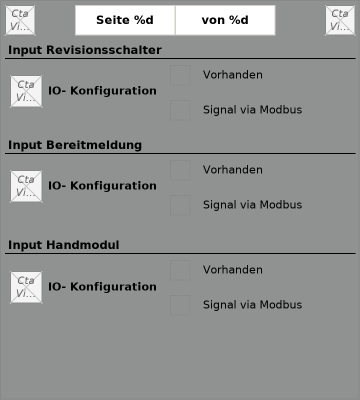
VISUALIZATION StellAntrieb_ParameterIO  // 360x400
VAR_INPUT
    ITF_STELLANTRIEBIN : ITF_STELLANTRIEB;
END_VAR
VAR
    uiPage  :   UINT;
    uiMin   :   UINT    := 0;
    uiMax   :   UINT    := 4;
END_VAR
    Frame (0,40 360x360), frame switch variable: uiPage
        shows StellAntrieb_ParameterIO0(ITF_STELLANTRIEBIN := ITF_STELLANTRIEBIN, ITF_RevSwitch_IN := ITF_STELLANTRIEBIN.proRevisionSwitch_ITF, ITF_Ready_IN := ITF_STELLANTRIEBIN.proActuatorReady_ITF, ITF_HandModul_IN := ITF_STELLANTRIEBIN.proHandModul_ITF)
        shows StellAntrieb_ParameterIO1(ITF_STELLANTRIEBIN := ITF_STELLANTRIEBIN, ITF_RückClosed_IN := ITF_STELLANTRIEBIN.proIsClosed_ITF)
        shows StellAntrieb_ParameterIO2(ITF_STELLANTRIEBIN := ITF_STELLANTRIEBIN, ITF_RückOffen_IN := ITF_STELLANTRIEBIN.proIsOpen_ITF)
        shows StellAntrieb_ParameterIO3(ITF_STELLANTRIEBIN := ITF_STELLANTRIEBIN, ITF_ActualPos_IN := ITF_STELLANTRIEBIN.proActualPosition_ITF)
        shows StellAntrieb_ParameterIO4(ITF_STELLANTRIEBIN := ITF_STELLANTRIEBIN, ITF_xOnAuf_IN := ITF_STELLANTRIEBIN.proOnOpen_ITF, ITF_xOnZu_IN := ITF_STELLANTRIEBIN.proOnClose_ITF, ITF_rOnY_IN := ITF_STELLANTRIEBIN.proOnY_ITF)
    Image (325,5 30x30), invisible if: uiPage = uiMax, image: CtaVisSymbols.ImagePool.arrow-right_square
        OnMouseClick: execute {
            uiPage := uiPage + 1;
            IF uiPage >= uiMax THEN
                uiPage := uiMax;
            END_IF;
        }
    Image (5,5 30x30), invisible if: uiPage = uiMin, image: CtaVisSymbols.ImagePool.arrow-left_square
        OnMouseClick: execute {
            uiPage := uiPage - 1;
            IF uiPage <= uiMin THEN
                uiPage := uiMin;
            END_IF;
        }
    Textfield (175,5 100x30), "von %d", text variable: uiMax
    Textfield (75,5 100x30), "Seite %d", text variable: uiPage
END_VISUALIZATION

// 40 Visualizations/POPUP/PARAMETER/StellAntrieb_IO/StellAntrieb_ParameterIO2
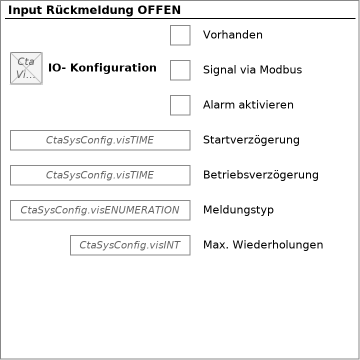
VISUALIZATION StellAntrieb_ParameterIO2  // 360x360
VAR_INPUT
    ITF_STELLANTRIEBIN 	:	ITF_STELLANTRIEB;
	ITF_RückOffen_IN	:	CtaSysIO.ITF_IO;
END_VAR
    Label (5,0 350x20), "Input Rückmeldung OFFEN"
    Frame (170,25 20x20)
        shows CtaSysConfig.visBOOL(visfbBOOLIn := ITF_STELLANTRIEBIN.p_scInStellAtRükOpen_fbxEnable)
    Label (200,25 150x20), "Vorhanden"
    Frame (170,60 20x20)
        shows CtaSysConfig.visBOOL(visfbBOOLIn := ITF_STELLANTRIEBIN.p_scInStellAtRükOpen_fbxInputMb)
    Label (200,60 150x20), "Signal via Modbus"
    Frame (170,95 20x20)
        shows CtaSysConfig.visBOOL(visfbBOOLIn := ITF_STELLANTRIEBIN.p_scInStellAtRükOpen_fbxDoesAlarm)
    Label (200,95 150x20), "Alarm aktivieren"
    Frame (10,130 180x20)
        shows CtaSysConfig.visTIME(visfbTIMEIn := ITF_STELLANTRIEBIN.p_scInStellAtRükOpen_fbtDelayStart)
    Label (200,130 150x20), "Startverzögerung"
    Label (200,165 150x20), "Betriebsverzögerung"
    Frame (10,165 180x20)
        shows CtaSysConfig.visTIME(visfbTIMEIn := ITF_STELLANTRIEBIN.p_scInStellAtRükOpen_fbtDelayRun)
    Label (200,200 150x20), "Meldungstyp"
    Label (200,235 150x20), "Max. Wiederholungen"
    Line (5,18) (355,18)
    Frame (10,200 180x20), text list: 'CtaAppReport.txtLibAp99_2enTypeOfAck', text index: CtaSysConfig.fcGetEnumerationId(ITF_STELLANTRIEBIN.p_scInStellAtRükOpen_fbiTypeOfAck)
        shows CtaSysConfig.visENUMERATION(visfbENUIn := ITF_STELLANTRIEBIN.p_scInStellAtRükOpen_fbiTypeOfAck)
    Frame (70,235 120x20)
        shows CtaSysConfig.visINT(visfbINTIn := ITF_STELLANTRIEBIN.p_scInStellAtRükOpen_fbiMaxErrorRetryAllowed)
    Image (10,52 32x32), invisible if: ITF_RückOffen_IN = 0, image: CtaVisSymbols.ImagePool.build
        OnMouseDown:  Dialog=StellAntrieb_POPUP_IO_ITF, Parameters={ITF_IO_IN: ITF_RückOffen_IN}, OpenModal=True, OpenCentered=True
    Label (45,58 120x20), "IO- Konfiguration", invisible if: ITF_RückOffen_IN = 0
END_VISUALIZATION

// 40 Visualizations/POPUP/PARAMETER/StellAntrieb_IO/StellAntrieb_ParameterIO3
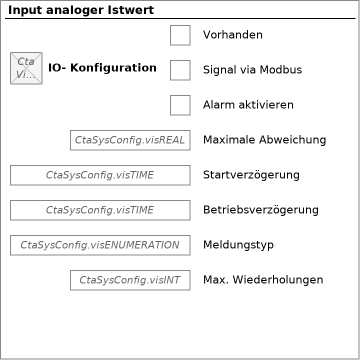
VISUALIZATION StellAntrieb_ParameterIO3  // 360x360
VAR_INPUT
    ITF_STELLANTRIEBIN 	:	ITF_STELLANTRIEB;
	ITF_ActualPos_IN	:	CtaSysIO.ITF_IO;
END_VAR
    Label (5,0 350x20), "Input analoger Istwert"
    Frame (170,25 20x20)
        shows CtaSysConfig.visBOOL(visfbBOOLIn := ITF_STELLANTRIEBIN.p_scInStellAtActualPosition_fbxEnable)
    Label (200,25 150x20), "Vorhanden"
    Frame (170,60 20x20)
        shows CtaSysConfig.visBOOL(visfbBOOLIn := ITF_STELLANTRIEBIN.p_scInStellAtActualPosition_fbxInputMb)
    Label (200,60 150x20), "Signal via Modbus"
    Frame (170,95 20x20)
        shows CtaSysConfig.visBOOL(visfbBOOLIn := ITF_STELLANTRIEBIN.p_scInStellAtActualPosition_fbxDoesAlarm)
    Label (200,95 150x20), "Alarm aktivieren"
    Frame (10,165 180x20)
        shows CtaSysConfig.visTIME(visfbTIMEIn := ITF_STELLANTRIEBIN.p_scInStellAtActualPosition_fbtDelayStart)
    Label (200,165 150x20), "Startverzögerung"
    Label (200,200 150x20), "Betriebsverzögerung"
    Frame (10,200 180x20)
        shows CtaSysConfig.visTIME(visfbTIMEIn := ITF_STELLANTRIEBIN.p_scInStellAtActualPosition_fbtDelayRun)
    Frame (70,130 120x20)
        shows CtaSysConfig.visREAL(visfbREALIn := ITF_STELLANTRIEBIN.p_scInStellAtActualPosition_fbrMaxDiff, stPhysikalischeEinheit := '%')
    Label (200,130 150x20), "Maximale Abweichung"
    Label (200,235 150x20), "Meldungstyp"
    Label (200,270 150x20), "Max. Wiederholungen"
    Line (5,18) (355,18)
    Frame (10,235 180x20), text list: 'CtaAppReport.txtLibAp99_2enTypeOfAck', text index: CtaSysConfig.fcGetEnumerationId(ITF_STELLANTRIEBIN.p_scInStellAtActualPosition_fbiTypeOfAck)
        shows CtaSysConfig.visENUMERATION(visfbENUIn := ITF_STELLANTRIEBIN.p_scInStellAtActualPosition_fbiTypeOfAck)
    Frame (70,270 120x20)
        shows CtaSysConfig.visINT(visfbINTIn := ITF_STELLANTRIEBIN.p_scInStellAtActualPosition_fbiMaxErrorRetryAllowed)
    Label (45,58 120x20), "IO- Konfiguration", invisible if: ITF_ActualPos_IN = 0
    Image (10,52 32x32), invisible if: ITF_ActualPos_IN = 0, image: CtaVisSymbols.ImagePool.build
        OnMouseDown:  Dialog=StellAntrieb_POPUP_IO_ITF, Parameters={ITF_IO_IN: ITF_ActualPos_IN}, OpenModal=True, OpenCentered=True
END_VISUALIZATION

// 40 Visualizations/POPUP/PARAMETER/StellAntrieb_InfluxDb/StellAntrieb_ParameterInfluxDb
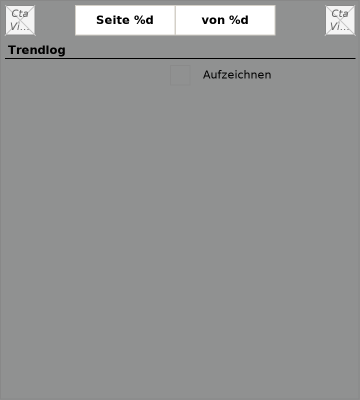
VISUALIZATION StellAntrieb_ParameterInfluxDb  // 360x400
VAR_INPUT
    ITF_STELLANTRIEBIN : ITF_STELLANTRIEB;
END_VAR
VAR
    uiPage  :   UINT;
    uiMin   :   UINT    := 0;
    uiMax   :   UINT    := 0;
END_VAR
    Image (5,5 30x30), invisible if: uiPage = uiMin, image: CtaVisSymbols.ImagePool.arrow-left_square
        OnMouseClick: execute {
            uiPage := uiPage - 1;
            IF uiPage <= uiMin THEN
                uiPage := uiMin;
            END_IF;
        }
    Image (325,5 30x30), invisible if: uiPage = uiMax, image: CtaVisSymbols.ImagePool.arrow-right_square
        OnMouseClick: execute {
            uiPage := uiPage + 1;
            IF uiPage >= uiMax THEN
                uiPage := uiMax;
            END_IF;
        }
    Frame (0,40 360x360), frame switch variable: uiPage
        shows StellAntrieb_ParameterInfluxDb0(ITF_STELLANTRIEBIN := ITF_STELLANTRIEBIN)
        shows AT_ParameterIO1(ITF_Parameter := ITF_Parameter)
        pReferences[0]: ITF_Parameter=ITF_Parameter
    Textfield (75,5 100x30), "Seite %d", text variable: uiPage
    Textfield (175,5 100x30), "von %d", text variable: uiMax
END_VISUALIZATION

// 40 Visualizations/POPUP/PARAMETER/StellAntrieb_InfluxDb/StellAntrieb_ParameterInfluxDb0
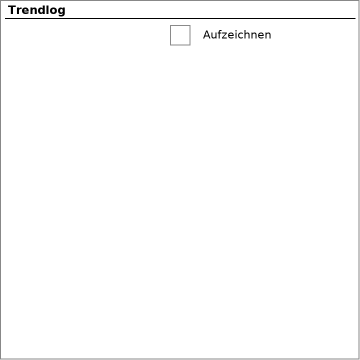
VISUALIZATION StellAntrieb_ParameterInfluxDb0  // 360x360
VAR_INPUT
    ITF_STELLANTRIEBIN : ITF_STELLANTRIEB;
END_VAR
    Frame (170,25 20x20)
        shows CtaSysConfig.visBOOL(visfbBOOLIn := ITF_STELLANTRIEBIN.p_scInfluxDb_fbxEnable)
    Label (200,25 150x20), "Aufzeichnen"
    Label (5,0 350x20), "Trendlog"
    Line (5,18) (355,18)
END_VISUALIZATION

// 40 Visualizations/POPUP/IO/StellAntrieb_IO0
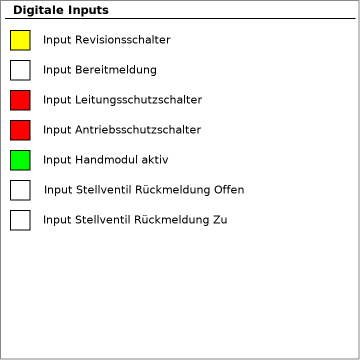
VISUALIZATION StellAntrieb_IO0  // 360x360
VAR_INPUT
    ITF_STELLANTRIEBIN    :   ITF_STELLANTRIEB;	
END_VAR
    Label (40,30 320x20), "Input Revisionsschalter", invisible if: ITF_STELLANTRIEBIN.proNotShowDI_RevisionSwitchOk
    Label (40,60 320x20), "Input Bereitmeldung", invisible if: ITF_STELLANTRIEBIN.proNotShowDI_Ready
    Rectangle (10,30 20x20), colour toggle: ITF_STELLANTRIEBIN.proGetDI_RevisionSwitchOK, invisible if: ITF_STELLANTRIEBIN.proNotShowDI_RevisionSwitchOk
    Rectangle (10,60 20x20), colour toggle: ITF_STELLANTRIEBIN.proGetDI_IsReady, invisible if: ITF_STELLANTRIEBIN.proNotShowDI_Ready
    Rectangle (10,90 20x20), colour toggle: ITF_STELLANTRIEBIN.proGetDI_FuseOK, invisible if: ITF_STELLANTRIEBIN.proNotShowDI_FuseOk
    Label (40,90 320x20), "Input Leitungsschutzschalter", invisible if: ITF_STELLANTRIEBIN.proNotShowDI_FuseOk
    Label (40,120 320x20), "Input Antriebsschutzschalter", invisible if: ITF_STELLANTRIEBIN.proNotShowDI_ActuatorFuseOk
    Rectangle (10,120 20x20), colour toggle: ITF_STELLANTRIEBIN.proGetDI_ActuatorFuseOk, invisible if: ITF_STELLANTRIEBIN.proNotShowDI_ActuatorFuseOk
    Label (40,150 320x20), "Input Handmodul aktiv", invisible if: ITF_STELLANTRIEBIN.proNotShowDI_ActuatorHand
    Rectangle (10,150 20x20), colour toggle: ITF_STELLANTRIEBIN.proGetDI_ActuatorHand, invisible if: ITF_STELLANTRIEBIN.proNotShowDI_ActuatorHand
    Label (10,0 350x20), "Digitale Inputs"
    Rectangle (10,210 20x20), colour toggle: ITF_STELLANTRIEBIN.proGetDI_RükIsClosed, invisible if: ITF_STELLANTRIEBIN.proNotShowDI_RükIsOpen
    Label (40,210 320x20), "Input Stellventil Rückmeldung Zu", invisible if: ITF_STELLANTRIEBIN.proNotShowDI_RükIsOpen
    Rectangle (10,180 20x20), colour toggle: ITF_STELLANTRIEBIN.proGetDI_RükIsOpen, invisible if: ITF_STELLANTRIEBIN.proNotShowDI_RükIsOpen
    Label (41,180 320x20), "Input Stellventil Rückmeldung Offen", invisible if: ITF_STELLANTRIEBIN.proNotShowDI_RükIsOpen
    Line (5,18) (355,18)
END_VISUALIZATION

// 40 Visualizations/POPUP/IO/StellAntrieb_IO
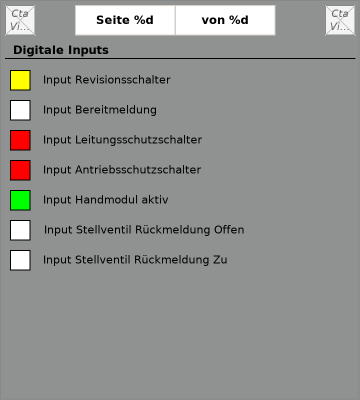
VISUALIZATION StellAntrieb_IO  // 360x400
VAR_INPUT
    ITF_STELLANTRIEBIN    :   ITF_STELLANTRIEB;	
END_VAR
VAR
    uiPage  :   UINT;
    uiMin   :   UINT    := 0;
    uiMax   :   UINT    := 1;
END_VAR
    Frame (0,40 360x360), frame switch variable: uiPage
        shows StellAntrieb_IO0(ITF_STELLANTRIEBIN := ITF_STELLANTRIEBIN)
        shows StellAntrieb_IO1(ITF_STELLANTRIEBIN := ITF_STELLANTRIEBIN)
        shows AT_ParameterIO2(ITF_Parameter := ITF_Parameter)
        shows AT_ParameterIO3(ITF_Parameter := ITF_Parameter)
    Image (325,5 30x30), invisible if: uiPage = uiMax, image: CtaVisSymbols.ImagePool.arrow-right_square
        OnMouseClick: execute {
            uiPage := uiPage + 1;
            IF uiPage >= uiMax THEN
                uiPage := uiMax;
            END_IF;
        }
    Image (5,5 30x30), invisible if: uiPage = uiMin, image: CtaVisSymbols.ImagePool.arrow-left_square
        OnMouseClick: execute {
            uiPage := uiPage - 1;
            IF uiPage <= uiMin THEN
                uiPage := uiMin;
            END_IF;
        }
    Textfield (175,5 100x30), "von %d", text variable: uiMax
    Textfield (75,5 100x30), "Seite %d", text variable: uiPage
END_VISUALIZATION

// 40 Visualizations/POPUP/IO/StellAntrieb_IO1
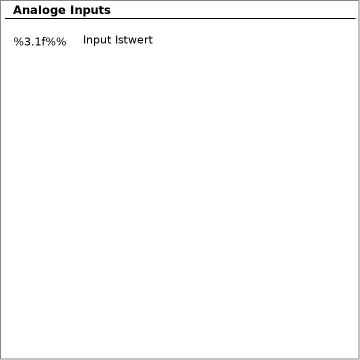
VISUALIZATION StellAntrieb_IO1  // 360x360
VAR_INPUT
    ITF_STELLANTRIEBIN    :   ITF_STELLANTRIEB;	
END_VAR
    Label (80,30 280x20), "Input Istwert", invisible if: ITF_STELLANTRIEBIN.proNotShowAI_ActualPosition
    Label (10,0 350x20), "Analoge Inputs"
    Textfield (10,32 60x20), "%3.1f%%", text variable: ITF_STELLANTRIEBIN.proGetAI_ActualPosition, invisible if: ITF_STELLANTRIEBIN.proNotShowAI_ActualPosition
    Line (5,18) (355,18)
END_VISUALIZATION

// 40 Visualizations/ICON/StellAntrieb_BASE/Ventile/DurchflussVentil/Motor_Left/ML_Durchgang
VISUALIZATION ML_Durchgang  // 15x30
VAR_INPUT
	rProzent	:	REAL;
END_VAR
    Line (0,15) (8,15)
    Polygon (8,15) (15,0) (0,0)
    Polygon (8,15) (15,30) (0,30)
    Polygon (8,15) (15,0) (0,0)
        p1097714728: fcValveAnimation(rProzent,TRUE)
END_VISUALIZATION

// 40 Visualizations/ICON/StellAntrieb_BASE/Icons/Motor_Left/Icon_ML_AB_Down
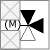
VISUALIZATION Icon_ML_AB_Down  // 50x50
VAR_INPUT
    ITF_STELLANTRIEB_IN   :   ITF_STELLANTRIEB;	
END_VAR
    Frame (5,17 15x15)
        shows Motor(ITF_STELLANTRIEB_IN := ITF_STELLANTRIEB_IN)
    Frame (20,10 22x30)
        shows ML_Ventil_AB_Down(rProzent := ITF_STELLANTRIEB_IN.proOnY)
    Image (0,0 20x20), invisible if: NOT ITF_STELLANTRIEB_IN.proIsWarning, image: CtaVisSymbols.ImagePool.CtaWarning
    Image (0,30 20x20), invisible if: NOT ITF_STELLANTRIEB_IN.proIsHandOnOrOff, image: CtaVisSymbols.ImagePool.front_hand_Yellow
    Image (0,30 20x20), invisible if: NOT ITF_STELLANTRIEB_IN.proHandOff, image: CtaVisSymbols.ImagePool.front_hand_Yellow_Off
END_VISUALIZATION

// 40 Visualizations/ICON/StellAntrieb_BASE/Ventile/DreiWegVentil/Motor_Above/MA_Ventil_AB_L
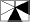
VISUALIZATION MA_Ventil_AB_L  // 30x22
VAR_INPUT
	rProzent	:	REAL;
END_VAR
    Polygon (0,0) (15,7) (0,15)
    Polygon (15,7) (22,22) (7,22)
    Polygon (15,7) (30,0) (30,15)
    Line (15,7) (15,0)
    Polygon (15,7) (30,0) (30,15)
        p1097714728: fcValveAnimation(rProzent,TRUE)
    Polygon (15,7) (22,22) (7,22)
        p1097714728: fcValveAnimation(rProzent,FALSE)
END_VISUALIZATION

// 40 Visualizations/ICON/StellAntrieb_BASE/Ventile/DreiWegVentil/Motor_Above/MA_Ventil_Verteiler
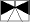
VISUALIZATION MA_Ventil_Verteiler  // 30x22
VAR_INPUT
	rProzent	:	REAL;
END_VAR
    Polygon (0,0) (15,7) (0,15)
    Polygon (15,7) (22,22) (7,22)
    Polygon (15,7) (30,0) (30,15)
    Line (15,7) (15,0)
    Polygon (15,7) (30,0) (30,15)
        p1097714728: fcValveAnimation(rProzent,FALSE)
    Polygon (0,0) (15,7) (0,15)
        p1097714728: fcValveAnimation(rProzent,TRUE)
END_VISUALIZATION

// 40 Visualizations/ICON/StellAntrieb_BASE/Ventile/DreiWegVentil/Motor_Above/MA_Ventil_AB_R
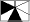
VISUALIZATION MA_Ventil_AB_R  // 30x22
VAR_INPUT
	rProzent	:	REAL;
END_VAR
    Polygon (0,0) (15,7) (0,15)
    Polygon (15,7) (22,22) (7,22)
    Polygon (15,7) (30,0) (30,15)
    Line (15,7) (15,0)
    Polygon (15,7) (22,22) (7,22)
        p1097714728: fcValveAnimation(rProzent,FALSE)
    Polygon (0,0) (15,7) (0,15)
        p1097714728: fcValveAnimation(rProzent,TRUE)
END_VISUALIZATION

// 40 Visualizations/ICON/StellAntrieb_BASE/Ventile/DreiWegVentil/Motor_Left/ML_Ventil_AB_Down
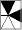
VISUALIZATION ML_Ventil_AB_Down  // 22x30
VAR_INPUT
	rProzent	:	REAL;
END_VAR
    Polygon (8,15) (15,0) (0,0)
    Polygon (8,15) (15,30) (0,30)
    Polygon (8,15) (23,8) (23,23)
    Line (0,15) (9,15)
    Polygon (8,15) (23,8) (23,23)
        p1097714728: fcValveAnimation(rProzent,False)
    Polygon (8,15) (15,0) (0,0)
        p1097714728: fcValveAnimation(rProzent,TRUE)
END_VISUALIZATION

// 40 Visualizations/ICON/StellAntrieb_BASE/Ventile/DreiWegVentil/Motor_Left/ML_Ventil_Verteiler
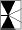
VISUALIZATION ML_Ventil_Verteiler  // 22x30
VAR_INPUT
	rProzent	:	REAL;
END_VAR
    Polygon (8,15) (15,0) (0,0)
    Polygon (8,15) (15,30) (0,30)
    Polygon (8,15) (23,8) (23,23)
    Line (0,15) (9,15)
    Polygon (8,15) (15,0) (0,0)
        p1097714728: fcValveAnimation(rProzent,FALSE)
    Polygon (8,15) (15,30) (0,30)
        p1097714728: fcValveAnimation(rProzent,TRUE)
END_VISUALIZATION

// 40 Visualizations/ICON/StellAntrieb_BASE/Ventile/DreiWegVentil/Motor_Left/ML_Ventil_AB_Up
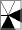
VISUALIZATION ML_Ventil_AB_Up  // 22x30
VAR_INPUT
	rProzent	:	REAL;
END_VAR
    Polygon (8,15) (15,0) (0,0)
    Polygon (8,15) (15,30) (0,30)
    Polygon (8,15) (23,8) (23,23)
    Line (0,15) (9,15)
    Polygon (8,15) (23,8) (23,23)
        p1097714728: fcValveAnimation(rProzent,FALSE)
    Polygon (8,15) (15,30) (0,30)
        p1097714728: fcValveAnimation(rProzent,TRUE)
END_VISUALIZATION

// 40 Visualizations/ICON/StellAntrieb_BASE/Ventile/DreiWegVentil/Motor_Below/MB_Ventil_AB_L
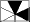
VISUALIZATION MB_Ventil_AB_L  // 30x22
VAR_INPUT
	rProzent	:	REAL;
END_VAR
    Polygon (15,15) (22,0) (7,0)
    Polygon (0,7) (15,14) (0,22)
    Polygon (15,14) (30,7) (30,22)
    Line (15,22) (15,13)
    Polygon (15,14) (30,7) (30,22)
        p1097714728: fcValveAnimation(rProzent,TRUE)
    Polygon (15,14) (22,0) (7,0)
        p1097714728: fcValveAnimation(rProzent,FALSE)
END_VISUALIZATION

// 40 Visualizations/ICON/StellAntrieb_BASE/Ventile/DreiWegVentil/Motor_Below/MB_Ventil_Verteiler
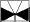
VISUALIZATION MB_Ventil_Verteiler  // 30x22
VAR_INPUT
	rProzent	:	REAL;
END_VAR
    Polygon (15,15) (22,0) (7,0)
    Polygon (0,7) (15,14) (0,22)
    Polygon (15,14) (30,7) (30,22)
    Line (15,22) (15,13)
    Polygon (15,14) (30,7) (30,22)
        p1097714728: fcValveAnimation(rProzent,TRUE)
    Polygon (0,7) (15,14) (0,22)
        p1097714728: fcValveAnimation(rProzent,FALSE)
END_VISUALIZATION

// 40 Visualizations/ICON/StellAntrieb_BASE/Ventile/DreiWegVentil/Motor_Below/MB_Ventil_AB_R
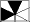
VISUALIZATION MB_Ventil_AB_R  // 30x22
VAR_INPUT
	rProzent	:	REAL;
END_VAR
    Polygon (15,15) (22,0) (7,0)
    Polygon (0,7) (15,14) (0,22)
    Polygon (15,14) (30,7) (30,22)
    Line (15,22) (15,13)
    Polygon (0,7) (15,14) (0,22)
        p1097714728: fcValveAnimation(rProzent,TRUE)
    Polygon (15,15) (22,0) (7,0)
        p1097714728: fcValveAnimation(rProzent,FALSE)
END_VISUALIZATION

// 40 Visualizations/ICON/StellAntrieb_BASE/Ventile/DreiWegVentil/Motor_Right/MR_Ventil_AB_Up
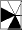
VISUALIZATION MR_Ventil_AB_Up  // 22x30
VAR_INPUT
	rProzent	:	REAL;
END_VAR
    Polygon (15,15) (22,0) (7,0)
    Polygon (15,15) (22,30) (7,30)
    Polygon (15,15) (0,7) (0,22)
    Line (14,15) (22,15)
    Polygon (15,15) (0,7) (0,22)
        p1097714728: fcValveAnimation(rProzent,FALSE)
    Polygon (15,15) (22,30) (7,30)
        p1097714728: fcValveAnimation(rProzent,TRUE)
END_VISUALIZATION

// 40 Visualizations/ICON/StellAntrieb_BASE/Ventile/DreiWegVentil/Motor_Right/MR_Ventil_Verteiler
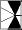
VISUALIZATION MR_Ventil_Verteiler  // 22x30
VAR_INPUT
	rProzent	:	REAL;
END_VAR
    Polygon (15,15) (22,0) (7,0)
    Polygon (15,15) (22,30) (7,30)
    Polygon (15,15) (0,7) (0,22)
    Line (14,15) (22,15)
    Polygon (15,15) (22,0) (7,0)
        p1097714728: fcValveAnimation(rProzent,FALSE)
    Polygon (15,15) (22,30) (7,30)
        p1097714728: fcValveAnimation(rProzent,TRUE)
END_VISUALIZATION

// 40 Visualizations/ICON/StellAntrieb_BASE/Ventile/DreiWegVentil/Motor_Right/MR_Ventil_AB_Down
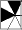
VISUALIZATION MR_Ventil_AB_Down  // 22x30
VAR_INPUT
	rProzent	:	REAL;
END_VAR
    Polygon (15,15) (22,0) (7,0)
    Polygon (15,15) (22,30) (7,30)
    Polygon (15,15) (0,7) (0,22)
    Line (14,15) (22,15)
    Polygon (15,15) (22,0) (7,0)
        p1097714728: fcValveAnimation(rProzent,FALSE)
    Polygon (15,15) (0,7) (0,22)
        p1097714728: fcValveAnimation(rProzent,TRUE)
END_VISUALIZATION

// 40 Visualizations/ICON/StellAntrieb_BASE/Ventile/DurchflussVentil/Motor_Right/MR_Durchgang
VISUALIZATION MR_Durchgang  // 15x30
VAR_INPUT
	rProzent	:	REAL;
END_VAR
    Line (7,15) (15,15)
    Polygon (7,15) (15,0) (0,0)
    Polygon (7,15) (15,30) (0,30)
    Polygon (7,15) (15,0) (0,0)
        p1097714728: fcValveAnimation(rProzent,TRUE)
END_VISUALIZATION

// 40 Visualizations/ICON/StellAntrieb_BASE/Ventile/DurchflussVentil/Motor_Below/MB_Durchgang
VISUALIZATION MB_Durchgang  // 30x15
VAR_INPUT
	rProzent	:	REAL;
END_VAR
    Line (15,7) (15,15)
    Polygon (0,0) (15,7) (0,15)
    Polygon (15,7) (30,0) (30,15)
    Polygon (0,0) (15,7) (0,15)
        p1097714728: fcValveAnimation(rProzent,TRUE)
END_VISUALIZATION

// 40 Visualizations/ICON/StellAntrieb_BASE/Ventile/DurchflussVentil/Motor_Above/MA_Durchgang
VISUALIZATION MA_Durchgang  // 30x15
VAR_INPUT
	rProzent	:	REAL;
END_VAR
    Line (15,0) (15,7)
    Polygon (0,0) (15,7) (0,15)
    Polygon (15,7) (30,0) (30,15)
    Polygon (0,0) (15,7) (0,15)
        p1097714728: fcValveAnimation(rProzent,TRUE)
END_VISUALIZATION

// 40 Visualizations/ICON/StellAntrieb_BASE/Icons/Motor_Left/Icon_ML_AB_Up
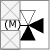
VISUALIZATION Icon_ML_AB_Up  // 50x50
VAR_INPUT
    ITF_STELLANTRIEB_IN   :   ITF_STELLANTRIEB;	
END_VAR
    Frame (5,17 15x15)
        shows Motor(ITF_STELLANTRIEB_IN := ITF_STELLANTRIEB_IN)
    Frame (20,10 22x30)
        shows ML_Ventil_AB_Up(rProzent := ITF_STELLANTRIEB_IN.proOnY)
    Image (0,0 20x20), invisible if: NOT ITF_STELLANTRIEB_IN.proIsWarning, image: CtaVisSymbols.ImagePool.CtaWarning
    Image (0,30 20x20), invisible if: NOT ITF_STELLANTRIEB_IN.proIsHandOnOrOff, image: CtaVisSymbols.ImagePool.front_hand_Yellow
    Image (0,30 20x20), invisible if: NOT ITF_STELLANTRIEB_IN.proHandOff, image: CtaVisSymbols.ImagePool.front_hand_Yellow_Off
END_VISUALIZATION

// 40 Visualizations/ICON/StellAntrieb_BASE/Icons/Motor_Left/Icon_ML_Verteiler
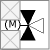
VISUALIZATION Icon_ML_Verteiler  // 50x50
VAR_INPUT
    ITF_STELLANTRIEB_IN   :   ITF_STELLANTRIEB;	
END_VAR
    Frame (5,17 15x15)
        shows Motor(ITF_STELLANTRIEB_IN := ITF_STELLANTRIEB_IN)
    Frame (20,10 22x30)
        shows ML_Ventil_Verteiler(rProzent := ITF_STELLANTRIEB_IN.proOnY)
    Image (0,0 20x20), invisible if: NOT ITF_STELLANTRIEB_IN.proIsWarning, image: CtaVisSymbols.ImagePool.CtaWarning
    Image (0,30 20x20), invisible if: NOT ITF_STELLANTRIEB_IN.proIsHandOnOrOff, image: CtaVisSymbols.ImagePool.front_hand_Yellow
    Image (0,30 20x20), invisible if: NOT ITF_STELLANTRIEB_IN.proHandOff, image: CtaVisSymbols.ImagePool.front_hand_Yellow_Off
END_VISUALIZATION

// 40 Visualizations/ICON/StellAntrieb_BASE/Icons/Motor_Left/Icon_ML_Durchfluss
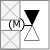
VISUALIZATION Icon_ML_Durchfluss  // 50x50
VAR_INPUT
    ITF_STELLANTRIEB_IN   :   ITF_STELLANTRIEB;	
END_VAR
    Frame (9,17 15x15)
        shows Motor(ITF_STELLANTRIEB_IN := ITF_STELLANTRIEB_IN)
    Frame (24,10 15x30)
        shows ML_Durchgang(rProzent := ITF_STELLANTRIEB_IN.proOnY)
    Image (0,0 20x20), invisible if: NOT ITF_STELLANTRIEB_IN.proIsWarning, image: CtaVisSymbols.ImagePool.CtaWarning
    Image (0,30 20x20), invisible if: NOT ITF_STELLANTRIEB_IN.proIsHandOnOrOff, image: CtaVisSymbols.ImagePool.front_hand_Yellow
    Image (0,30 20x20), invisible if: NOT ITF_STELLANTRIEB_IN.proHandOff, image: CtaVisSymbols.ImagePool.front_hand_Yellow_Off
END_VISUALIZATION

// 40 Visualizations/ICON/StellAntrieb_BASE/Icons/Motor_Right/Icon_MR_AB_Down
